# EPICS substitutions: apps/CaenHVApp/db/CaenHV_Test.substitutions
file "db/HVgroup.template" {
pattern
    {P,         H}
    {CAEN403,   36}
}

file "db/AS503_Chan.template" {
pattern
    {P,         H,      V}
    {CAEN403,   36,     0}
    {CAEN403,   36,     1}
    {CAEN403,   36,     2}
    {CAEN403,   36,     3}
    {CAEN403,   36,     4}
    {CAEN403,   36,     5}
    {CAEN403,   36,     6}
    {CAEN403,   36,     7}
    {CAEN403,   36,     8}
    {CAEN403,   36,     9}
    {CAEN403,   36,     10}
    {CAEN403,   36,     11}
    {CAEN403,   36,     12}
    {CAEN403,   36,     13}
    {CAEN403,   36,     14}
    {CAEN403,   36,     15}
    {CAEN403,   36,     16}
    {CAEN403,   36,     17}
    {CAEN403,   36,     18}
    {CAEN403,   36,     19}
    {CAEN403,   36,     20}
    {CAEN403,   36,     21}
    {CAEN403,   36,     22}
    {CAEN403,   36,     23}
    {CAEN403,   36,     24}
    {CAEN403,   36,     25}
    {CAEN403,   36,     26}
    {CAEN403,   36,     27}
    {CAEN403,   36,     28}
    {CAEN403,   36,     29}
    {CAEN403,   36,     30}
    {CAEN403,   36,     31}
    {CAEN403,   36,     32}
    {CAEN403,   36,     33}
    {CAEN403,   36,     34}
    {CAEN403,   36,     35}
    {CAEN403,   36,     36}
    {CAEN403,   36,     37}
    {CAEN403,   36,     38}
    {CAEN403,   36,     39}
    {CAEN403,   36,     40}
    {CAEN403,   36,     41}
    {CAEN403,   36,     42}
    {CAEN403,   36,     43}
    {CAEN403,   36,     44}
    {CAEN403,   36,     45}
    {CAEN403,   36,     46}
    {CAEN403,   36,     47}
    {CAEN403,   36,     48}
    {CAEN403,   36,     49}
    {CAEN403,   36,     50}
    {CAEN403,   36,     51}
    {CAEN403,   36,     52}
    {CAEN403,   36,     53}
    {CAEN403,   36,     54}
    {CAEN403,   36,     55}
    {CAEN403,   36,     56}
    {CAEN403,   36,     57}
    {CAEN403,   36,     58}
    {CAEN403,   36,     59}
    {CAEN403,   36,     60}
    {CAEN403,   36,     61}
    {CAEN403,   36,     62}
    {CAEN403,   36,     63}
}
